# EPICS substitutions: mc04/db/motor.substitutions
file "db/motor.db"
{

# ADDR ---> axis #
# NOTE ---> 2 asyn ports: 1) lowel comms ("P0"), and 2) Motor Record ("motor")
pattern
{ P,             M,               MOTOR,   PORT,    ADDR, DESC,     DTYP }
{ "XF:23ID1-BI", "{Diag:2-Ax:Y}Mtr", 	  "motor", "PO",    1,  "Diag:2 y-axis", asynMotor }
}
